TYPE TcoPlsPaletizator_Control_v_1_x_x EXTENDS TcoCore.TcoStruct:
STRUCT

		
END_STRUCT
END_TYPE

(* stored: Version 1.1.0.1
   DUT TcoPlsPaletizator_Control_v_1_x_x: Id {302a5062-e0e4-49ac-b8b0-24da27bdb1ef} *)
